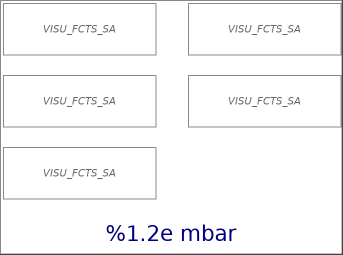
VISUALIZATION SA_POMP_ENCEINTE  // 343x255
VAR_IN_OUT
	m_Input_PRG:		BLOCK_PRG_POMPAGE;
	m_Input_Jauge:		BLOCK_BCG450_ETHERCAT;
END_VAR
    Rectangle (0,0 343x255)
    Frame (3,75 153x52)
        shows VISU_FCTS_SA(m_Input_ID_XML := 0, m_Input_UserRight := PRG_USER.ACTU_USER.FONCTION_SA, m_Input_Operation := m_Input_PRG.POMPAGE.OP_Pompage_Sec)
    Frame (3,3 153x52)
        shows VISU_FCTS_SA(m_Input_ID_XML := 1, m_Input_UserRight := PRG_USER.ACTU_USER.FONCTION_SA, m_Input_Operation := m_Input_PRG.POMPAGE.OP_Marche_Pompes)
    Frame (188,3 153x52)
        shows VISU_FCTS_SA(m_Input_ID_XML := 2, m_Input_UserRight := PRG_USER.ACTU_USER.FONCTION_SA, m_Input_Operation := m_Input_PRG.POMPAGE.OP_Arret_Pompes)
    Frame (188,75 153x52)
        shows VISU_FCTS_SA(m_Input_ID_XML := 3, m_Input_UserRight := PRG_USER.ACTU_USER.FONCTION_SA, m_Input_Operation := m_Input_PRG.POMPAGE.OP_Isolement)
    Frame (3,147 153x52)
        shows VISU_FCTS_SA(m_Input_ID_XML := 4, m_Input_UserRight := PRG_USER.ACTU_USER.FONCTION_SA, m_Input_Operation := m_Input_PRG.POMPAGE.OP_Ventilation)
    Rectangle (80,219 182x29), "%1.2e mbar", text variable: m_Input_Jauge.STATE_Pression
END_VISUALIZATION

(* stored: Version 1.1.0.1, ProductVersion 3.1.4024.10
   Visu SA_POMP_ENCEINTE: Id {b151c58d-5a62-4c48-9cff-b3007a758cd5} *)
